// TIA Portal V17 export
// export: Created 2025-03-05T08:00:05.3597551Z, ExportSetting WithDefaults, DisplayName Totally Integrated Automation Portal, DisplayVersion V17 Update 8, DisplayName TIA Portal Openness, DisplayVersion V17 Update 8, DisplayName TIA Portal Version Control Interface, DisplayVersion V17, DisplayName SINAMICS Startdrive Advanced, DisplayVersion V17 SP2, DisplayName SINAMICS Startdrive G110M, G120, G120C, G120D, G120P, G115D, DisplayVersion V17 SP2, DisplayName SINAMICS Startdrive G130, G150, S120, S150, SINAMICS MV, S210, DisplayVersion V17 SP2, DisplayName STEP 7 Professional, DisplayVersion V17 Update 8, DisplayName SINUMERIK ONE STEP 7 Toolbox, DisplayVersion V17 Update 12, DisplayName SINUMERIK 840D sl STEP 7 Toolbox, DisplayVersion V17 Update 12, DisplayName STEP 7 Safety, DisplayVersion V17 Update 6, DisplayName WinCC Advanced, DisplayVersion V17 Update 8
FUNCTION "FC2038_CALIBRATION_CYCLE" : Void   // FC2038, LAD
{ S7_Optimized_Access := 'TRUE' }
VERSION : 0.1
// stored: AutoNumber false, IsIECCheckEnabled false, SetENOAutomatically false, UDAEnableTagReadback false
   VAR_TEMP
      O_BYTE_0 : Struct   // OPTIONS BYTE 0
         MANUAL_LOAD_SELECTOR : Bool;   // MANUAL LOAD SELECTOR OPTION
      END_STRUCT;
   END_VAR
   VAR CONSTANT
      FC_NUMBER : Int := 2038;
   END_VAR
   VAR_TEMP   // added for the SCL form of the ladder/FBD networks
      _w1 : Bool;
      _w2 : Bool;
   END_VAR
BEGIN

REGION Network 1: MANUAL LOAD SELECTOR OPTION
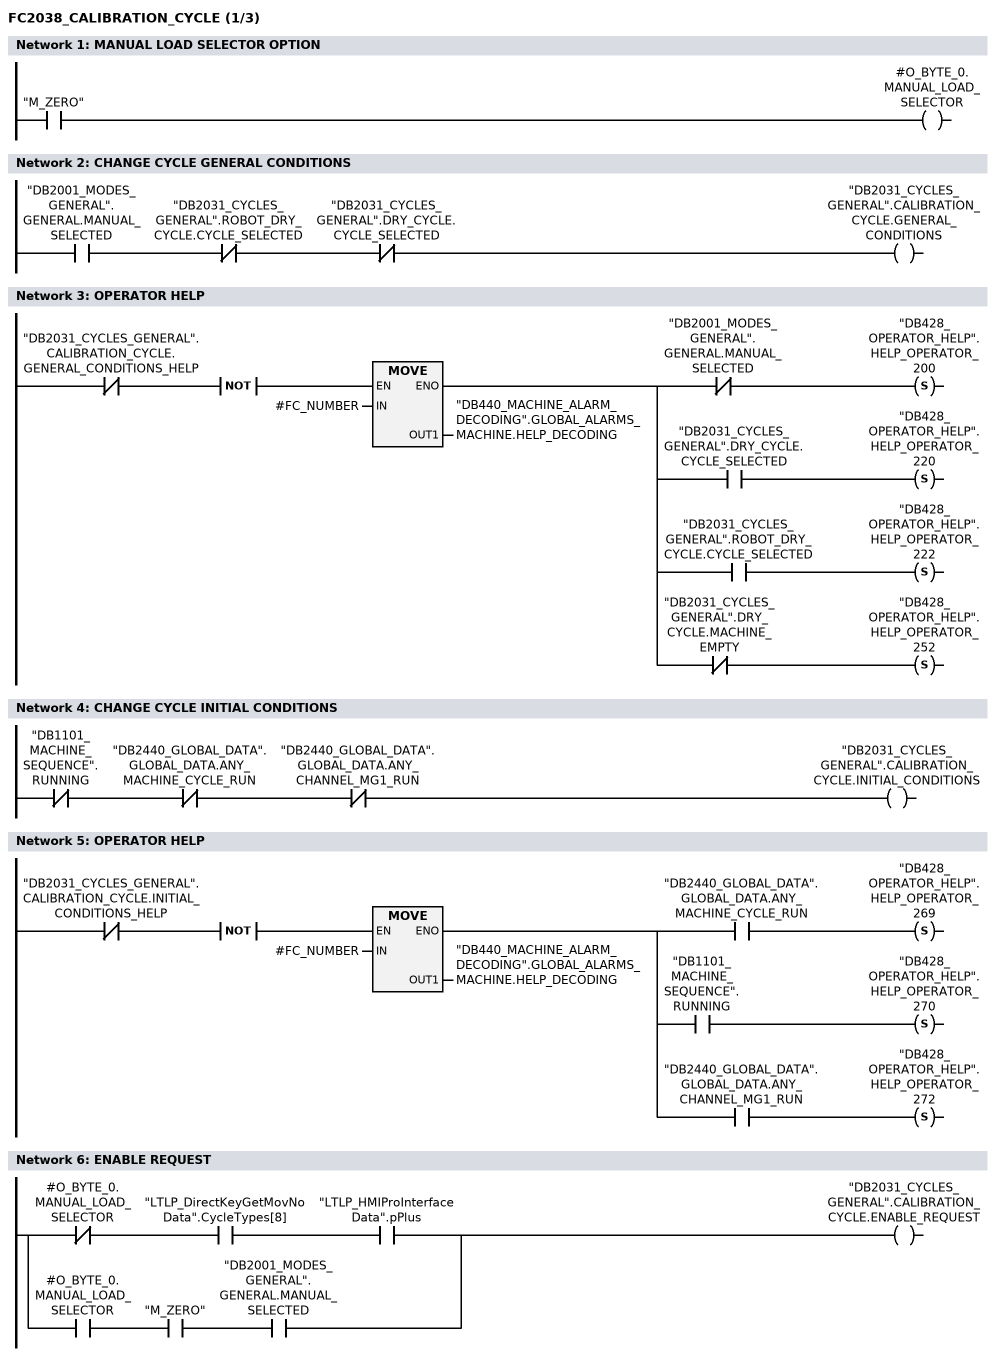
   RUNG wire#powerrail
      Contact( "M_ZERO" )
      Coil( #O_BYTE_0.MANUAL_LOAD_SELECTOR )
   END_RUNG
   // the same network as SCL:
   #O_BYTE_0.MANUAL_LOAD_SELECTOR := "M_ZERO";
END_REGION

REGION Network 2: CHANGE CYCLE GENERAL CONDITIONS
   RUNG wire#powerrail
      Contact( "DB2001_MODES_GENERAL".GENERAL.MANUAL_SELECTED )
      I_Contact( "DB2031_CYCLES_GENERAL".ROBOT_DRY_CYCLE.CYCLE_SELECTED )
      I_Contact( "DB2031_CYCLES_GENERAL".DRY_CYCLE.CYCLE_SELECTED )
      Coil( "DB2031_CYCLES_GENERAL".CALIBRATION_CYCLE.GENERAL_CONDITIONS )
   END_RUNG
   // the same network as SCL:
   "DB2031_CYCLES_GENERAL".CALIBRATION_CYCLE.GENERAL_CONDITIONS := "DB2001_MODES_GENERAL".GENERAL.MANUAL_SELECTED AND NOT "DB2031_CYCLES_GENERAL".ROBOT_DRY_CYCLE.CYCLE_SELECTED AND NOT "DB2031_CYCLES_GENERAL".DRY_CYCLE.CYCLE_SELECTED;
END_REGION

REGION Network 3: OPERATOR HELP
   RUNG wire#powerrail
      I_Contact( "DB2031_CYCLES_GENERAL".CALIBRATION_CYCLE.GENERAL_CONDITIONS_HELP )
      Not()
      { S7_GenerateENO := "TRUE" } Move(in := #FC_NUMBER, out1 => "DB440_MACHINE_ALARM_DECODING".GLOBAL_ALARMS_MACHINE.HELP_DECODING)
      wire#w1
      I_Contact( "DB2001_MODES_GENERAL".GENERAL.MANUAL_SELECTED )
      S_Coil( "DB428_OPERATOR_HELP".HELP_OPERATOR_200 )
   END_RUNG
   RUNG wire#w1
      Contact( "DB2031_CYCLES_GENERAL".DRY_CYCLE.CYCLE_SELECTED )
      S_Coil( "DB428_OPERATOR_HELP".HELP_OPERATOR_220 )
   END_RUNG
   RUNG wire#w1
      Contact( "DB2031_CYCLES_GENERAL".ROBOT_DRY_CYCLE.CYCLE_SELECTED )
      S_Coil( "DB428_OPERATOR_HELP".HELP_OPERATOR_222 )
   END_RUNG
   RUNG wire#w1
      I_Contact( "DB2031_CYCLES_GENERAL".DRY_CYCLE.MACHINE_EMPTY )
      S_Coil( "DB428_OPERATOR_HELP".HELP_OPERATOR_252 )
   END_RUNG
   // the same network as SCL:
   // ENO of a box is taken as its EN; it also drops when the box reports an error
   #_w1 := NOT (NOT "DB2031_CYCLES_GENERAL".CALIBRATION_CYCLE.GENERAL_CONDITIONS_HELP);
   IF #_w1 THEN "DB440_MACHINE_ALARM_DECODING".GLOBAL_ALARMS_MACHINE.HELP_DECODING := #FC_NUMBER; END_IF;
   IF #_w1 AND NOT "DB2001_MODES_GENERAL".GENERAL.MANUAL_SELECTED THEN
       "DB428_OPERATOR_HELP".HELP_OPERATOR_200 := TRUE;
   END_IF;
   IF #_w1 AND "DB2031_CYCLES_GENERAL".DRY_CYCLE.CYCLE_SELECTED THEN
       "DB428_OPERATOR_HELP".HELP_OPERATOR_220 := TRUE;
   END_IF;
   IF #_w1 AND "DB2031_CYCLES_GENERAL".ROBOT_DRY_CYCLE.CYCLE_SELECTED THEN
       "DB428_OPERATOR_HELP".HELP_OPERATOR_222 := TRUE;
   END_IF;
   IF #_w1 AND NOT "DB2031_CYCLES_GENERAL".DRY_CYCLE.MACHINE_EMPTY THEN
       "DB428_OPERATOR_HELP".HELP_OPERATOR_252 := TRUE;
   END_IF;
END_REGION

REGION Network 4: CHANGE CYCLE INITIAL CONDITIONS
   RUNG wire#powerrail
      I_Contact( "DB1101_MACHINE_SEQUENCE".RUNNING )
      I_Contact( "DB2440_GLOBAL_DATA".GLOBAL_DATA.ANY_MACHINE_CYCLE_RUN )
      I_Contact( "DB2440_GLOBAL_DATA".GLOBAL_DATA.ANY_CHANNEL_MG1_RUN )
      Coil( "DB2031_CYCLES_GENERAL".CALIBRATION_CYCLE.INITIAL_CONDITIONS )
   END_RUNG
   // the same network as SCL:
   "DB2031_CYCLES_GENERAL".CALIBRATION_CYCLE.INITIAL_CONDITIONS := NOT "DB1101_MACHINE_SEQUENCE".RUNNING AND NOT "DB2440_GLOBAL_DATA".GLOBAL_DATA.ANY_MACHINE_CYCLE_RUN AND NOT "DB2440_GLOBAL_DATA".GLOBAL_DATA.ANY_CHANNEL_MG1_RUN;
END_REGION

REGION Network 5: OPERATOR HELP
   RUNG wire#powerrail
      I_Contact( "DB2031_CYCLES_GENERAL".CALIBRATION_CYCLE.INITIAL_CONDITIONS_HELP )
      Not()
      { S7_GenerateENO := "TRUE" } Move(in := #FC_NUMBER, out1 => "DB440_MACHINE_ALARM_DECODING".GLOBAL_ALARMS_MACHINE.HELP_DECODING)
      wire#w1
      Contact( "DB2440_GLOBAL_DATA".GLOBAL_DATA.ANY_MACHINE_CYCLE_RUN )
      S_Coil( "DB428_OPERATOR_HELP".HELP_OPERATOR_269 )
   END_RUNG
   RUNG wire#w1
      Contact( "DB1101_MACHINE_SEQUENCE".RUNNING )
      S_Coil( "DB428_OPERATOR_HELP".HELP_OPERATOR_270 )
   END_RUNG
   RUNG wire#w1
      Contact( "DB2440_GLOBAL_DATA".GLOBAL_DATA.ANY_CHANNEL_MG1_RUN )
      S_Coil( "DB428_OPERATOR_HELP".HELP_OPERATOR_272 )
   END_RUNG
   // the same network as SCL:
   // ENO of a box is taken as its EN; it also drops when the box reports an error
   #_w1 := NOT (NOT "DB2031_CYCLES_GENERAL".CALIBRATION_CYCLE.INITIAL_CONDITIONS_HELP);
   IF #_w1 THEN "DB440_MACHINE_ALARM_DECODING".GLOBAL_ALARMS_MACHINE.HELP_DECODING := #FC_NUMBER; END_IF;
   IF #_w1 AND "DB2440_GLOBAL_DATA".GLOBAL_DATA.ANY_MACHINE_CYCLE_RUN THEN
       "DB428_OPERATOR_HELP".HELP_OPERATOR_269 := TRUE;
   END_IF;
   IF #_w1 AND "DB1101_MACHINE_SEQUENCE".RUNNING THEN
       "DB428_OPERATOR_HELP".HELP_OPERATOR_270 := TRUE;
   END_IF;
   IF #_w1 AND "DB2440_GLOBAL_DATA".GLOBAL_DATA.ANY_CHANNEL_MG1_RUN THEN
       "DB428_OPERATOR_HELP".HELP_OPERATOR_272 := TRUE;
   END_IF;
END_REGION

REGION Network 6: ENABLE REQUEST
   RUNG wire#powerrail
      I_Contact( #O_BYTE_0.MANUAL_LOAD_SELECTOR )
      Contact( "LTLP_DirectKeyGetMovNoData".CycleTypes[8] )
      Contact( "LTLP_HMIProInterfaceData".pPlus )
      wire#w1
      Coil( "DB2031_CYCLES_GENERAL".CALIBRATION_CYCLE.ENABLE_REQUEST )
   END_RUNG
   RUNG wire#powerrail
      Contact( #O_BYTE_0.MANUAL_LOAD_SELECTOR )
      Contact( "M_ZERO" )
      Contact( "DB2001_MODES_GENERAL".GENERAL.MANUAL_SELECTED )
   END_RUNG wire#w1
   // the same network as SCL:
   "DB2031_CYCLES_GENERAL".CALIBRATION_CYCLE.ENABLE_REQUEST := (NOT #O_BYTE_0.MANUAL_LOAD_SELECTOR AND "LTLP_DirectKeyGetMovNoData".CycleTypes[8] AND "LTLP_HMIProInterfaceData".pPlus) OR (#O_BYTE_0.MANUAL_LOAD_SELECTOR AND "M_ZERO" AND "DB2001_MODES_GENERAL".GENERAL.MANUAL_SELECTED);
END_REGION

REGION Network 7: DISABLE REQUEST
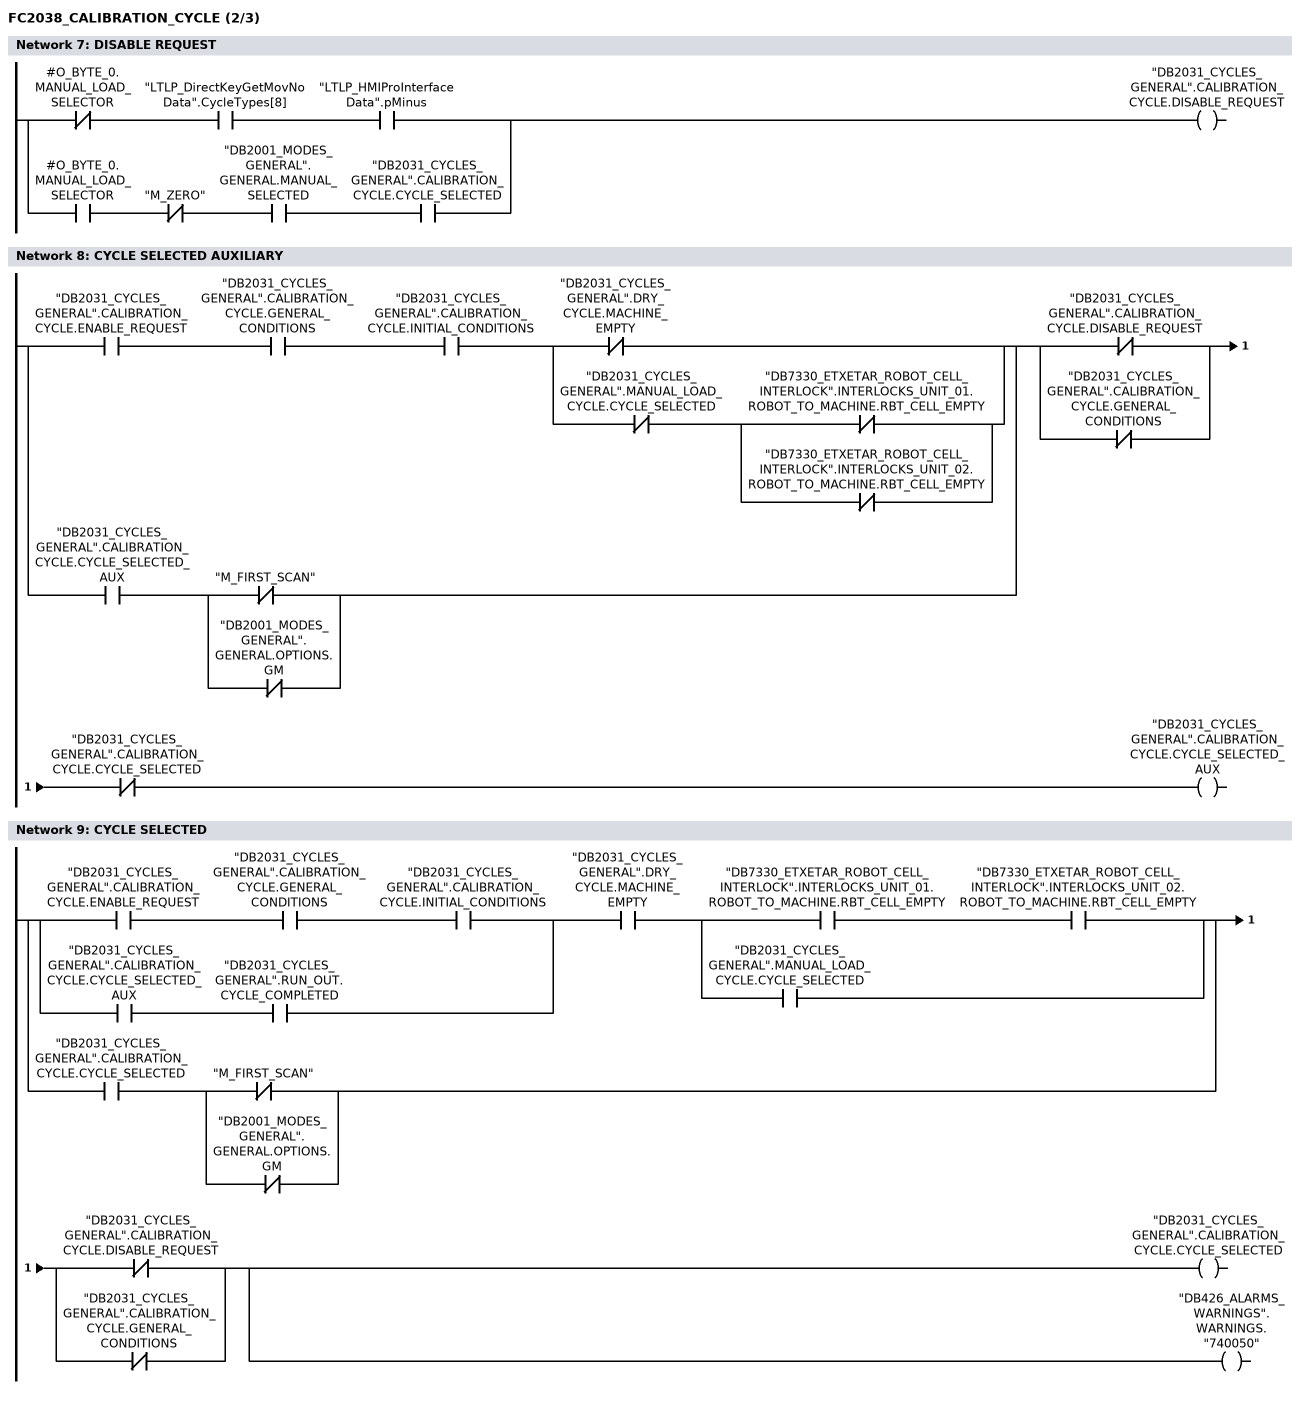
   RUNG wire#powerrail
      I_Contact( #O_BYTE_0.MANUAL_LOAD_SELECTOR )
      Contact( "LTLP_DirectKeyGetMovNoData".CycleTypes[8] )
      Contact( "LTLP_HMIProInterfaceData".pMinus )
      wire#w1
      Coil( "DB2031_CYCLES_GENERAL".CALIBRATION_CYCLE.DISABLE_REQUEST )
   END_RUNG
   RUNG wire#powerrail
      Contact( #O_BYTE_0.MANUAL_LOAD_SELECTOR )
      I_Contact( "M_ZERO" )
      Contact( "DB2001_MODES_GENERAL".GENERAL.MANUAL_SELECTED )
      Contact( "DB2031_CYCLES_GENERAL".CALIBRATION_CYCLE.CYCLE_SELECTED )
   END_RUNG wire#w1
   // the same network as SCL:
   "DB2031_CYCLES_GENERAL".CALIBRATION_CYCLE.DISABLE_REQUEST := (NOT #O_BYTE_0.MANUAL_LOAD_SELECTOR AND "LTLP_DirectKeyGetMovNoData".CycleTypes[8] AND "LTLP_HMIProInterfaceData".pMinus) OR (#O_BYTE_0.MANUAL_LOAD_SELECTOR AND NOT "M_ZERO" AND "DB2001_MODES_GENERAL".GENERAL.MANUAL_SELECTED AND "DB2031_CYCLES_GENERAL".CALIBRATION_CYCLE.CYCLE_SELECTED);
END_REGION

REGION Network 8: CYCLE SELECTED AUXILIARY
   RUNG wire#powerrail
      Contact( "DB2031_CYCLES_GENERAL".CALIBRATION_CYCLE.ENABLE_REQUEST )
      Contact( "DB2031_CYCLES_GENERAL".CALIBRATION_CYCLE.GENERAL_CONDITIONS )
      Contact( "DB2031_CYCLES_GENERAL".CALIBRATION_CYCLE.INITIAL_CONDITIONS )
      wire#w1
      I_Contact( "DB2031_CYCLES_GENERAL".DRY_CYCLE.MACHINE_EMPTY )
      wire#w2
      I_Contact( "DB2031_CYCLES_GENERAL".CALIBRATION_CYCLE.DISABLE_REQUEST )
      wire#w5
      I_Contact( "DB2031_CYCLES_GENERAL".CALIBRATION_CYCLE.CYCLE_SELECTED )
      Coil( "DB2031_CYCLES_GENERAL".CALIBRATION_CYCLE.CYCLE_SELECTED_AUX )
   END_RUNG
   RUNG wire#w1
      I_Contact( "DB2031_CYCLES_GENERAL".MANUAL_LOAD_CYCLE.CYCLE_SELECTED )
      wire#w3
      I_Contact( "DB7330_ETXETAR_ROBOT_CELL_INTERLOCK".INTERLOCKS_UNIT_01.ROBOT_TO_MACHINE.RBT_CELL_EMPTY )
   END_RUNG wire#w2
   RUNG wire#w3
      I_Contact( "DB7330_ETXETAR_ROBOT_CELL_INTERLOCK".INTERLOCKS_UNIT_02.ROBOT_TO_MACHINE.RBT_CELL_EMPTY )
   END_RUNG wire#w2
   RUNG wire#powerrail
      Contact( "DB2031_CYCLES_GENERAL".CALIBRATION_CYCLE.CYCLE_SELECTED_AUX )
      wire#w4
      I_Contact( "M_FIRST_SCAN" )
   END_RUNG wire#w2
   RUNG wire#w4
      I_Contact( "DB2001_MODES_GENERAL".GENERAL.OPTIONS.GM )
   END_RUNG wire#w2
   RUNG wire#w2
      I_Contact( "DB2031_CYCLES_GENERAL".CALIBRATION_CYCLE.GENERAL_CONDITIONS )
   END_RUNG wire#w5
   // the same network as SCL:
   "DB2031_CYCLES_GENERAL".CALIBRATION_CYCLE.CYCLE_SELECTED_AUX := (("DB2031_CYCLES_GENERAL".CALIBRATION_CYCLE.ENABLE_REQUEST AND "DB2031_CYCLES_GENERAL".CALIBRATION_CYCLE.GENERAL_CONDITIONS AND "DB2031_CYCLES_GENERAL".CALIBRATION_CYCLE.INITIAL_CONDITIONS AND (NOT "DB2031_CYCLES_GENERAL".DRY_CYCLE.MACHINE_EMPTY OR (NOT "DB2031_CYCLES_GENERAL".MANUAL_LOAD_CYCLE.CYCLE_SELECTED AND (NOT "DB7330_ETXETAR_ROBOT_CELL_INTERLOCK".INTERLOCKS_UNIT_01.ROBOT_TO_MACHINE.RBT_CELL_EMPTY OR NOT "DB7330_ETXETAR_ROBOT_CELL_INTERLOCK".INTERLOCKS_UNIT_02.ROBOT_TO_MACHINE.RBT_CELL_EMPTY)))) OR ("DB2031_CYCLES_GENERAL".CALIBRATION_CYCLE.CYCLE_SELECTED_AUX AND (NOT "M_FIRST_SCAN" OR NOT "DB2001_MODES_GENERAL".GENERAL.OPTIONS.GM))) AND (NOT "DB2031_CYCLES_GENERAL".CALIBRATION_CYCLE.DISABLE_REQUEST OR NOT "DB2031_CYCLES_GENERAL".CALIBRATION_CYCLE.GENERAL_CONDITIONS) AND NOT "DB2031_CYCLES_GENERAL".CALIBRATION_CYCLE.CYCLE_SELECTED;
END_REGION

REGION Network 9: CYCLE SELECTED
   RUNG wire#powerrail
      Contact( "DB2031_CYCLES_GENERAL".CALIBRATION_CYCLE.ENABLE_REQUEST )
      Contact( "DB2031_CYCLES_GENERAL".CALIBRATION_CYCLE.GENERAL_CONDITIONS )
      Contact( "DB2031_CYCLES_GENERAL".CALIBRATION_CYCLE.INITIAL_CONDITIONS )
      wire#w1
      Contact( "DB2031_CYCLES_GENERAL".DRY_CYCLE.MACHINE_EMPTY )
      wire#w2
      Contact( "DB7330_ETXETAR_ROBOT_CELL_INTERLOCK".INTERLOCKS_UNIT_01.ROBOT_TO_MACHINE.RBT_CELL_EMPTY )
      Contact( "DB7330_ETXETAR_ROBOT_CELL_INTERLOCK".INTERLOCKS_UNIT_02.ROBOT_TO_MACHINE.RBT_CELL_EMPTY )
      wire#w3
      I_Contact( "DB2031_CYCLES_GENERAL".CALIBRATION_CYCLE.DISABLE_REQUEST )
      wire#w5
      Coil( "DB2031_CYCLES_GENERAL".CALIBRATION_CYCLE.CYCLE_SELECTED )
   END_RUNG
   RUNG wire#powerrail
      Contact( "DB2031_CYCLES_GENERAL".CALIBRATION_CYCLE.CYCLE_SELECTED_AUX )
      Contact( "DB2031_CYCLES_GENERAL".RUN_OUT.CYCLE_COMPLETED )
   END_RUNG wire#w1
   RUNG wire#w2
      Contact( "DB2031_CYCLES_GENERAL".MANUAL_LOAD_CYCLE.CYCLE_SELECTED )
   END_RUNG wire#w3
   RUNG wire#powerrail
      Contact( "DB2031_CYCLES_GENERAL".CALIBRATION_CYCLE.CYCLE_SELECTED )
      wire#w4
      I_Contact( "M_FIRST_SCAN" )
   END_RUNG wire#w3
   RUNG wire#w4
      I_Contact( "DB2001_MODES_GENERAL".GENERAL.OPTIONS.GM )
   END_RUNG wire#w3
   RUNG wire#w3
      I_Contact( "DB2031_CYCLES_GENERAL".CALIBRATION_CYCLE.GENERAL_CONDITIONS )
   END_RUNG wire#w5
   RUNG wire#w5
      Coil( "DB426_ALARMS_WARNINGS".WARNINGS."740050" )
   END_RUNG
   // the same network as SCL:
   "DB2031_CYCLES_GENERAL".CALIBRATION_CYCLE.CYCLE_SELECTED := (((("DB2031_CYCLES_GENERAL".CALIBRATION_CYCLE.ENABLE_REQUEST AND "DB2031_CYCLES_GENERAL".CALIBRATION_CYCLE.GENERAL_CONDITIONS AND "DB2031_CYCLES_GENERAL".CALIBRATION_CYCLE.INITIAL_CONDITIONS) OR ("DB2031_CYCLES_GENERAL".CALIBRATION_CYCLE.CYCLE_SELECTED_AUX AND "DB2031_CYCLES_GENERAL".RUN_OUT.CYCLE_COMPLETED)) AND "DB2031_CYCLES_GENERAL".DRY_CYCLE.MACHINE_EMPTY AND (("DB7330_ETXETAR_ROBOT_CELL_INTERLOCK".INTERLOCKS_UNIT_01.ROBOT_TO_MACHINE.RBT_CELL_EMPTY AND "DB7330_ETXETAR_ROBOT_CELL_INTERLOCK".INTERLOCKS_UNIT_02.ROBOT_TO_MACHINE.RBT_CELL_EMPTY) OR "DB2031_CYCLES_GENERAL".MANUAL_LOAD_CYCLE.CYCLE_SELECTED)) OR ("DB2031_CYCLES_GENERAL".CALIBRATION_CYCLE.CYCLE_SELECTED AND (NOT "M_FIRST_SCAN" OR NOT "DB2001_MODES_GENERAL".GENERAL.OPTIONS.GM))) AND (NOT "DB2031_CYCLES_GENERAL".CALIBRATION_CYCLE.DISABLE_REQUEST OR NOT "DB2031_CYCLES_GENERAL".CALIBRATION_CYCLE.GENERAL_CONDITIONS);
   "DB426_ALARMS_WARNINGS".WARNINGS."740050" := "DB2031_CYCLES_GENERAL".CALIBRATION_CYCLE.CYCLE_SELECTED;
END_REGION

REGION Network 10: STOP END OF CYCLE WARNING
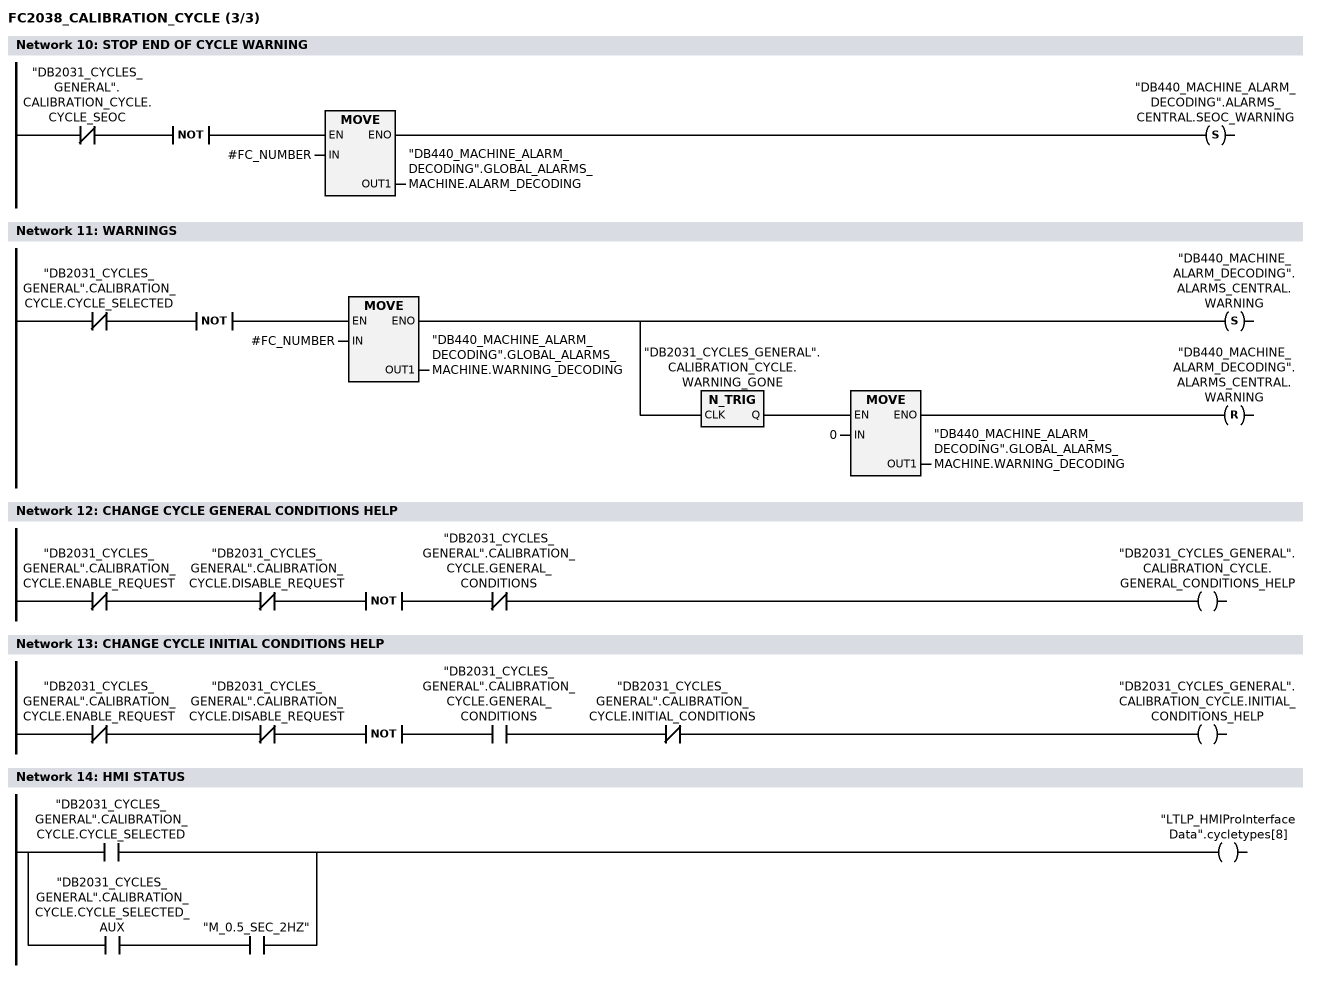
   RUNG wire#powerrail
      I_Contact( "DB2031_CYCLES_GENERAL".CALIBRATION_CYCLE.CYCLE_SEOC )
      Not()
      { S7_GenerateENO := "TRUE" } Move(in := #FC_NUMBER, out1 => "DB440_MACHINE_ALARM_DECODING".GLOBAL_ALARMS_MACHINE.ALARM_DECODING)
      S_Coil( "DB440_MACHINE_ALARM_DECODING".ALARMS_CENTRAL.SEOC_WARNING )
   END_RUNG
   // the same network as SCL:
   // ENO of a box is taken as its EN; it also drops when the box reports an error
   IF NOT (NOT "DB2031_CYCLES_GENERAL".CALIBRATION_CYCLE.CYCLE_SEOC) THEN
       "DB440_MACHINE_ALARM_DECODING".GLOBAL_ALARMS_MACHINE.ALARM_DECODING := #FC_NUMBER;
       "DB440_MACHINE_ALARM_DECODING".ALARMS_CENTRAL.SEOC_WARNING := TRUE;
   END_IF;
END_REGION

REGION Network 11: WARNINGS
   RUNG wire#powerrail
      I_Contact( "DB2031_CYCLES_GENERAL".CALIBRATION_CYCLE.CYCLE_SELECTED )
      Not()
      Move(in := #FC_NUMBER, out1 => "DB440_MACHINE_ALARM_DECODING".GLOBAL_ALARMS_MACHINE.WARNING_DECODING)
      wire#w1
      S_Coil( "DB440_MACHINE_ALARM_DECODING".ALARMS_CENTRAL.WARNING )
   END_RUNG
   RUNG wire#w1
      N_Trig( "DB2031_CYCLES_GENERAL".CALIBRATION_CYCLE.WARNING_GONE )
      Move(in := 0, out1 => "DB440_MACHINE_ALARM_DECODING".GLOBAL_ALARMS_MACHINE.WARNING_DECODING)
      R_Coil( "DB440_MACHINE_ALARM_DECODING".ALARMS_CENTRAL.WARNING )
   END_RUNG
   // the same network as SCL:
   #_w1 := NOT (NOT "DB2031_CYCLES_GENERAL".CALIBRATION_CYCLE.CYCLE_SELECTED);
   IF #_w1 THEN
       "DB440_MACHINE_ALARM_DECODING".GLOBAL_ALARMS_MACHINE.WARNING_DECODING := #FC_NUMBER;
       "DB440_MACHINE_ALARM_DECODING".ALARMS_CENTRAL.WARNING := TRUE;
   END_IF;
   #_w2 := NOT #_w1 AND "DB2031_CYCLES_GENERAL".CALIBRATION_CYCLE.WARNING_GONE;   // falling edge
   "DB2031_CYCLES_GENERAL".CALIBRATION_CYCLE.WARNING_GONE := #_w1;
   IF #_w2 THEN
       "DB440_MACHINE_ALARM_DECODING".GLOBAL_ALARMS_MACHINE.WARNING_DECODING := 0;
       "DB440_MACHINE_ALARM_DECODING".ALARMS_CENTRAL.WARNING := FALSE;
   END_IF;
END_REGION

REGION Network 12: CHANGE CYCLE GENERAL CONDITIONS HELP
   RUNG wire#powerrail
      I_Contact( "DB2031_CYCLES_GENERAL".CALIBRATION_CYCLE.ENABLE_REQUEST )
      I_Contact( "DB2031_CYCLES_GENERAL".CALIBRATION_CYCLE.DISABLE_REQUEST )
      Not()
      I_Contact( "DB2031_CYCLES_GENERAL".CALIBRATION_CYCLE.GENERAL_CONDITIONS )
      Coil( "DB2031_CYCLES_GENERAL".CALIBRATION_CYCLE.GENERAL_CONDITIONS_HELP )
   END_RUNG
   // the same network as SCL:
   "DB2031_CYCLES_GENERAL".CALIBRATION_CYCLE.GENERAL_CONDITIONS_HELP := NOT (NOT "DB2031_CYCLES_GENERAL".CALIBRATION_CYCLE.ENABLE_REQUEST AND NOT "DB2031_CYCLES_GENERAL".CALIBRATION_CYCLE.DISABLE_REQUEST) AND NOT "DB2031_CYCLES_GENERAL".CALIBRATION_CYCLE.GENERAL_CONDITIONS;
END_REGION

REGION Network 13: CHANGE CYCLE INITIAL CONDITIONS HELP
   RUNG wire#powerrail
      I_Contact( "DB2031_CYCLES_GENERAL".CALIBRATION_CYCLE.ENABLE_REQUEST )
      I_Contact( "DB2031_CYCLES_GENERAL".CALIBRATION_CYCLE.DISABLE_REQUEST )
      Not()
      Contact( "DB2031_CYCLES_GENERAL".CALIBRATION_CYCLE.GENERAL_CONDITIONS )
      I_Contact( "DB2031_CYCLES_GENERAL".CALIBRATION_CYCLE.INITIAL_CONDITIONS )
      Coil( "DB2031_CYCLES_GENERAL".CALIBRATION_CYCLE.INITIAL_CONDITIONS_HELP )
   END_RUNG
   // the same network as SCL:
   "DB2031_CYCLES_GENERAL".CALIBRATION_CYCLE.INITIAL_CONDITIONS_HELP := NOT (NOT "DB2031_CYCLES_GENERAL".CALIBRATION_CYCLE.ENABLE_REQUEST AND NOT "DB2031_CYCLES_GENERAL".CALIBRATION_CYCLE.DISABLE_REQUEST) AND "DB2031_CYCLES_GENERAL".CALIBRATION_CYCLE.GENERAL_CONDITIONS AND NOT "DB2031_CYCLES_GENERAL".CALIBRATION_CYCLE.INITIAL_CONDITIONS;
END_REGION

REGION Network 14: HMI STATUS
   RUNG wire#powerrail
      Contact( "DB2031_CYCLES_GENERAL".CALIBRATION_CYCLE.CYCLE_SELECTED )
      wire#w1
      Coil( "LTLP_HMIProInterfaceData".cycletypes[8] )
   END_RUNG
   RUNG wire#powerrail
      Contact( "DB2031_CYCLES_GENERAL".CALIBRATION_CYCLE.CYCLE_SELECTED_AUX )
      Contact( "M_0.5_SEC_2HZ" )
   END_RUNG wire#w1
   // the same network as SCL:
   "LTLP_HMIProInterfaceData".cycletypes[8] := "DB2031_CYCLES_GENERAL".CALIBRATION_CYCLE.CYCLE_SELECTED OR ("DB2031_CYCLES_GENERAL".CALIBRATION_CYCLE.CYCLE_SELECTED_AUX AND "M_0.5_SEC_2HZ");
END_REGION
END_FUNCTION
